FUNCTION_BLOCK FB_PIDD (* PID with Bumpless Transfer and Anti-Reset Windup *)
  (* Standard: 61499-1-D.1 *)
  (* Version 0.1, 2001-04-21, JHC, Rockwell Automation, Laid out ECC. *)
  (* Version 0.0, 2000-04-29, JHC, Rockwell Automation *)
  (* Compiler header: package fb.rt.process; *)
  (* Compiler Java IBM VisualAge 3.0 *)
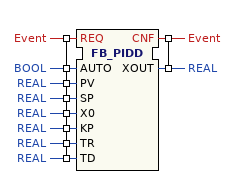
  EVENT_INPUT
    REQ WITH AUTO, PV, SP, X0, KP, TR, TD;
  END_EVENT
  EVENT_OUTPUT
    CNF WITH XOUT;
  END_EVENT
  VAR_INPUT
    AUTO : BOOL; (* 0-manual,1-automatic *)
    PV : REAL; (* Process variable,0-100 percent *)
    SP : REAL; (* Set Point,0-100 percent *)
    X0 : REAL; (* Manual Output Setting,0-100 percent *)
    KP : REAL; (* Proportionality Constant *)
    TR : REAL; (* Reset Time as Multiple of Sampling Period *)
    TD : REAL; (* Derivative Time Constant as Multiple of Sampling Period *)
  END_VAR
  VAR_OUTPUT
    XOUT : REAL; (* Manipulated Variable,0-100 percent *)
  END_VAR
  VAR
    WASAUTO : BOOL;
    ERROR : REAL;
    ITERM : REAL;
    DTERM : REAL;
    X1 : REAL;
    X2 : REAL;
    X3 : REAL;
  END_VAR
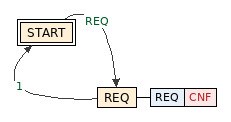
  EC_STATES
    START;
    REQ : REQ -> CNF;
  END_STATES
  EC_TRANSITIONS
    START TO REQ := REQ;
    REQ TO START := 1;
  END_TRANSITIONS
  ALGORITHM REQ IN ST:
ERROR:=PV-SP;

IF AUTO THEN

IF WASAUTO THEN

ITERM:=ITERM+ERROR/TR;

DTERM:=(3*(ERROR-X3)+X1-X2)/10*TD;

ELSE

ITERM:=(X0-ERROR)/KP;

DTERM:=0;

END_IF;

XOUT:=KP*(ERROR+ITERM+DTERM);

ELSE XOUT:=X0;

END_IF

X2:=X1;X1:=ERROR;

IF XOUT<0 THEN XOUT:=0;

ITERM:=ITERM-ERROR/TR;

ELSIF XOUT>100 THEN XOUT:=100;

ITERM:=ITERM-ERROR/TR;

END_IF;

WASAUTO:=AUTO;
  END_ALGORITHM
END_FUNCTION_BLOCK
